{attribute 'qualified_only'}
VAR_GLOBAL
END_VAR

(* stored: Version 1.1.0.1, ProductVersion 3.1.4024.12
   GVL gHMI: Id {4eac3206-c742-4329-a252-1f8d6893b0ff} *)
